// State handler: RESUMING
// Transient state — immediately signals → RUNNING.
// Add ramp-up logic here if needed in the future.
FUNCTION_BLOCK FB_State_Resuming
VAR_INPUT
    bExecute    : BOOL;
END_VAR
VAR_OUTPUT
    outCmd          : E_StateCmd := E_StateCmd.NONE;
    outEnable_Auto  : BOOL;
    outEnable_Man   : BOOL;
    outgvFault      : BOOL;
    outInit_VYHYBKY : BOOL;
    outInit_IMP_LEV : BOOL;
    outInit_IMP_PRA : BOOL;
END_VAR

IF NOT bExecute THEN
    outCmd          := E_StateCmd.NONE;
    outEnable_Auto  := FALSE;
    outEnable_Man   := FALSE;
    outgvFault      := FALSE;
    outInit_VYHYBKY := FALSE;
    outInit_IMP_LEV := FALSE;
    outInit_IMP_PRA := FALSE;
    RETURN;
END_IF

outEnable_Auto  := FALSE;
outEnable_Man   := FALSE;
outgvFault      := FALSE;
outInit_VYHYBKY := FALSE;
outInit_IMP_LEV := FALSE;
outInit_IMP_PRA := FALSE;

// Immediate transition
outCmd := E_StateCmd.TO_RUNNING;

END_FUNCTION_BLOCK

(* stored: Version 1.1.0.1, ProductVersion 3.1.4024.13
   POU FB_State_Resuming: Id {b1000006-0006-4000-8000-000000000006}, SpecialFunc None *)
